// TIA Portal V21 export
DATA_BLOCK "Dzieleniedb"   // DB3
{ S7_Optimized_Access := 'TRUE' }
   VAR
      z1 : Real;
      z2 : Real := 30.0;
      wynik : Real;
   END_VAR
BEGIN
END_DATA_BLOCK
